{attribute 'qualified_only'}
{attribute 'strict'}
TYPE E_ACTION_STATE :
(
	uninit := 0,
	ready,
	done1,
	done2,
	done3,
	done4,
	done5,
	done6,
	done7,
	done8,
	done9,
	done10,
	busy,
	error
);
END_TYPE

(* stored: Version 1.1.0.1, ProductVersion 3.1.4024.12
   DUT E_ACTION_STATE: Id {f0ae24b7-2532-46a6-91ee-eebf6871e145} *)
